// TIA Portal V20 export
DATA_BLOCK "CallInterfaceSignalsConv_BA10"   // DB347
// stored: InstanceOfName CallInterfaceSignalsConv, InstanceOfType FB
"CallInterfaceSignalsConv"
   // VAR_INPUT
   //    InterfaceTestMode : Bool := FALSE;
   // END_VAR
   // VAR_OUTPUT
   //    signalsS2R : "typeReelCutToStack";
   //    signalsR2S : "typeStackToReelCut";
   // END_VAR
   // VAR_IN_OUT
   //    CommS2R : Array[0..95] of Bool;
   //    CommR2S : Array[0..95] of Bool;
   //    InterfaceTestButton : "LER_SignalsInput";
   // END_VAR
   // VAR
   //    statWordBuffer_2 { S7_SetPoint := 'True'} : Array[0..5] of Word;
   //    statWordBuffer_1 : Array[0..5] of Word;
   // END_VAR
BEGIN
   signalsS2R.Load_Enable := FALSE;
   signalsS2R.Load_Complete_Comfirm := FALSE;
   signalsS2R.Cell_Data_Report := FALSE;
   signalsS2R.signal3 := FALSE;
   signalsS2R.signal4 := FALSE;
   signalsS2R.signal5 := FALSE;
   signalsS2R.signal6 := FALSE;
   signalsS2R.signal7 := FALSE;
   signalsS2R.signal8 := FALSE;
   signalsS2R.signal9 := FALSE;
   signalsS2R.signal10 := FALSE;
   signalsS2R.signal11 := FALSE;
   signalsS2R.signal12 := FALSE;
   signalsS2R.signal13 := FALSE;
   signalsS2R.signal14 := FALSE;
   signalsS2R.HeartBeat := FALSE;
   signalsS2R.signal16 := FALSE;
   signalsS2R.signal17 := FALSE;
   signalsS2R.signal18 := FALSE;
   signalsS2R.signal19 := FALSE;
   signalsS2R.signal20 := FALSE;
   signalsS2R.signal21 := FALSE;
   signalsS2R.signal22 := FALSE;
   signalsS2R.signal23 := FALSE;
   signalsS2R.signal24 := FALSE;
   signalsS2R.signal25 := FALSE;
   signalsS2R.signal26 := FALSE;
   signalsS2R.signal27 := FALSE;
   signalsS2R.signal28 := FALSE;
   signalsS2R.signal29 := FALSE;
   signalsS2R.signal30 := FALSE;
   signalsS2R.signal31 := FALSE;
   signalsS2R.signal32 := FALSE;
   signalsS2R.signal33 := FALSE;
   signalsS2R.signal34 := FALSE;
   signalsS2R.signal35 := FALSE;
   signalsS2R.signal36 := FALSE;
   signalsS2R.signal37 := FALSE;
   signalsS2R.signal38 := FALSE;
   signalsS2R.signal39 := FALSE;
   signalsS2R.signal40 := FALSE;
   signalsS2R.signal41 := FALSE;
   signalsS2R.signal42 := FALSE;
   signalsS2R.signal43 := FALSE;
   signalsS2R.signal44 := FALSE;
   signalsS2R.signal45 := FALSE;
   signalsS2R.signal46 := FALSE;
   signalsS2R.signal47 := FALSE;
   signalsS2R.signal48 := FALSE;
   signalsS2R.signal49 := FALSE;
   signalsS2R.signal50 := FALSE;
   signalsS2R.signal51 := FALSE;
   signalsS2R.signal52 := FALSE;
   signalsS2R.signal53 := FALSE;
   signalsS2R.signal54 := FALSE;
   signalsS2R.signal55 := FALSE;
   signalsS2R.signal56 := FALSE;
   signalsS2R.signal57 := FALSE;
   signalsS2R.signal58 := FALSE;
   signalsS2R.signal59 := FALSE;
   signalsS2R.signal60 := FALSE;
   signalsS2R.signal61 := FALSE;
   signalsS2R.signal62 := FALSE;
   signalsS2R.signal63 := FALSE;
   signalsS2R.signal64 := FALSE;
   signalsS2R.signal65 := FALSE;
   signalsS2R.signal66 := FALSE;
   signalsS2R.signal67 := FALSE;
   signalsS2R.signal68 := FALSE;
   signalsS2R.signal69 := FALSE;
   signalsS2R.signal70 := FALSE;
   signalsS2R.signal71 := FALSE;
   signalsS2R.signal72 := FALSE;
   signalsS2R.signal73 := FALSE;
   signalsS2R.signal74 := FALSE;
   signalsS2R.signal75 := FALSE;
   signalsS2R.signal76 := FALSE;
   signalsS2R.signal77 := FALSE;
   signalsS2R.signal78 := FALSE;
   signalsS2R.signal79 := FALSE;
   signalsS2R.signal80 := FALSE;
   signalsS2R.signal81 := FALSE;
   signalsS2R.signal82 := FALSE;
   signalsS2R.signal83 := FALSE;
   signalsS2R.signal84 := FALSE;
   signalsS2R.signal85 := FALSE;
   signalsS2R.signal86 := FALSE;
   signalsS2R.signal87 := FALSE;
   signalsS2R.signal88 := FALSE;
   signalsS2R.signal89 := FALSE;
   signalsS2R.signal90 := FALSE;
   signalsS2R.signal91 := FALSE;
   signalsS2R.signal92 := FALSE;
   signalsS2R.signal93 := FALSE;
   signalsS2R.signal94 := FALSE;
   signalsS2R.signal95 := FALSE;
   signalsR2S.Load_Requset := FALSE;
   signalsR2S.Load_Busy := FALSE;
   signalsR2S.Load_Complete := FALSE;
   signalsR2S.Cell_Data_Request := FALSE;
   signalsR2S.Cell_Data_Report_Ack := FALSE;
   signalsR2S.Cell_Data_Report_Nck := FALSE;
   signalsR2S.signal6 := FALSE;
   signalsR2S.signal7 := FALSE;
   signalsR2S.signal8 := FALSE;
   signalsR2S.signal9 := FALSE;
   signalsR2S.signal10 := FALSE;
   signalsR2S.signal11 := FALSE;
   signalsR2S.signal12 := FALSE;
   signalsR2S.signal13 := FALSE;
   signalsR2S.signal14 := FALSE;
   signalsR2S.HeartBeat := FALSE;
   signalsR2S.signal16 := FALSE;
   signalsR2S.signal17 := FALSE;
   signalsR2S.signal18 := FALSE;
   signalsR2S.signal19 := FALSE;
   signalsR2S.signal20 := FALSE;
   signalsR2S.signal21 := FALSE;
   signalsR2S.signal22 := FALSE;
   signalsR2S.signal23 := FALSE;
   signalsR2S.signal24 := FALSE;
   signalsR2S.signal25 := FALSE;
   signalsR2S.signal26 := FALSE;
   signalsR2S.signal27 := FALSE;
   signalsR2S.signal28 := FALSE;
   signalsR2S.signal29 := FALSE;
   signalsR2S.signal30 := FALSE;
   signalsR2S.signal31 := FALSE;
   signalsR2S.signal32 := FALSE;
   signalsR2S.signal33 := FALSE;
   signalsR2S.signal34 := FALSE;
   signalsR2S.signal35 := FALSE;
   signalsR2S.signal36 := FALSE;
   signalsR2S.signal37 := FALSE;
   signalsR2S.signal38 := FALSE;
   signalsR2S.signal39 := FALSE;
   signalsR2S.signal40 := FALSE;
   signalsR2S.signal41 := FALSE;
   signalsR2S.signal42 := FALSE;
   signalsR2S.signal43 := FALSE;
   signalsR2S.signal44 := FALSE;
   signalsR2S.signal45 := FALSE;
   signalsR2S.signal46 := FALSE;
   signalsR2S.signal47 := FALSE;
   signalsR2S.signal48 := FALSE;
   signalsR2S.signal49 := FALSE;
   signalsR2S.signal50 := FALSE;
   signalsR2S.signal51 := FALSE;
   signalsR2S.signal52 := FALSE;
   signalsR2S.signal53 := FALSE;
   signalsR2S.signal54 := FALSE;
   signalsR2S.signal55 := FALSE;
   signalsR2S.signal56 := FALSE;
   signalsR2S.signal57 := FALSE;
   signalsR2S.signal58 := FALSE;
   signalsR2S.signal59 := FALSE;
   signalsR2S.signal60 := FALSE;
   signalsR2S.signal61 := FALSE;
   signalsR2S.signal62 := FALSE;
   signalsR2S.signal63 := FALSE;
   signalsR2S.signal64 := FALSE;
   signalsR2S.signal65 := FALSE;
   signalsR2S.signal66 := FALSE;
   signalsR2S.signal67 := FALSE;
   signalsR2S.signal68 := FALSE;
   signalsR2S.signal69 := FALSE;
   signalsR2S.signal70 := FALSE;
   signalsR2S.signal71 := FALSE;
   signalsR2S.signal72 := FALSE;
   signalsR2S.signal73 := FALSE;
   signalsR2S.signal74 := FALSE;
   signalsR2S.signal75 := FALSE;
   signalsR2S.signal76 := FALSE;
   signalsR2S.signal77 := FALSE;
   signalsR2S.signal78 := FALSE;
   signalsR2S.signal79 := FALSE;
   signalsR2S.signal80 := FALSE;
   signalsR2S.signal81 := FALSE;
   signalsR2S.signal82 := FALSE;
   signalsR2S.signal83 := FALSE;
   signalsR2S.signal84 := FALSE;
   signalsR2S.signal85 := FALSE;
   signalsR2S.signal86 := FALSE;
   signalsR2S.signal87 := FALSE;
   signalsR2S.signal88 := FALSE;
   signalsR2S.signal89 := FALSE;
   signalsR2S.signal90 := FALSE;
   signalsR2S.signal91 := FALSE;
   signalsR2S.signal92 := FALSE;
   signalsR2S.signal93 := FALSE;
   signalsR2S.signal94 := FALSE;
   signalsR2S.signal95 := FALSE;
   statWordBuffer_2[0..5] := 16#0000;
   statWordBuffer_1[0..5] := 16#0000;
END_DATA_BLOCK
